TYPE ZCom :
STRUCT
  // module context
  App : ZApplication.ApplicationComPublish;
  Alarming : ZApplication.AlarmingCom;
  Messages : ZApplication.MessagingCom;
  
  // unit context
  Unit : ZComUnit;

END_STRUCT
END_TYPE

(* stored: Version 1.1.0.1
   DUT ZCom: Id {4ed7f0be-b2d7-40a9-9bfd-48b2eb3a875c} *)
